# EPICS autosave request: ADCore/ADApp/Db/NDPluginBase_settings.req
$(P)$(R)NDArrayPort
$(P)$(R)NDArrayAddress
$(P)$(R)EnableCallbacks
$(P)$(R)MinCallbackTime
$(P)$(R)BlockingCallbacks
$(P)$(R)NDAttributesFile
